// TIA Portal V16 export
// export: Created 2024-05-11T02:56:23.0061867Z, ExportSetting WithDefaults, DisplayName Totally Integrated Automation Portal, DisplayVersion V16, DisplayName TIA Portal Version Control Interface, DisplayVersion V16, DisplayName TIA Portal Openness, DisplayVersion V16, DisplayName STEP 7 Professional, DisplayVersion V16, DisplayName STEP 7 Safety, DisplayVersion V16, DisplayName WinCC Professional, DisplayVersion V16
FUNCTION_BLOCK "F100_Val"   // FB100, LAD
TITLE = 电磁阀控制，
{ S7_Optimized_Access := 'TRUE' }
VERSION : 0.1
// IW_ConMode    00= 双端实际传感器到位，10=出端虚拟到位，11=出双端虚拟到位，01=回端端虚拟到位，
// stored: AutoNumber false, IsIECCheckEnabled false, IsRetainMemResEnabled false, MemoryReserve 100, SetENOAutomatically false, UDAEnableTagReadback false
   VAR_INPUT
      I_AutoAdv : Bool;   // 自动出指令
      I_AutoRet : Bool;   // 自动回指令
      I_ManAdv : Bool;   // 手动出指令
      I_ManRet : Bool;   // 手动回指令
      I_AdvCond : Bool;   // 动作出条件
      I_RetCond : Bool;   // 动作回条件
      I_AdvLS : Bool;   // 伸出到位
      I_RetLS : Bool;   // 返回到位
      IW_AdvTime : Time;   // 出or虚拟延迟
      IW_RetTime : Time;   // 回or虚拟延迟
      IW_AdvTimeOver : Time;   // 伸出超时
      IW_RetTimeOver : Time;   // 返回超时
      I_FoBrRel : Bool;   // 刹车强制解除
      I_Rest : Bool;   // 异常复位
      I_ManMode : Bool;   // 手动模式
      IW_ConMode : UInt;   // 虚拟控制
   END_VAR
   VAR_OUTPUT
      Q_AdvEnd : Bool;   // 伸出到位延迟
      Q_RetEnd : Bool;   // 返回到位延迟
      Q_AdvLS : Bool;   // 伸出到位
      Q_RetLS : Bool;   // 返回到位
      Q_AdvSL : Bool;   // 伸出输出
      Q_RetSL : Bool;   // 返回输出
      Q_FoBraRel : Bool;   // 刹车解除输出
      Q_AdvTiOvErr { ExternalAccessible := 'False'; ExternalVisible := 'False'; ExternalWritable := 'False'} : Bool;   // 出动作超时故障
      Q_RetTiOvErr { ExternalAccessible := 'False'; ExternalVisible := 'False'; ExternalWritable := 'False'} : Bool;   // 回动作超时故障
      Q_SensorsErr : Bool;   // 到位传感器都ON故障
      Q_SenCroErr : Bool;   // 到位传感器交叉ON故障
   END_VAR
   VAR
      MT_AdvChK { ExternalAccessible := 'False'; ExternalVisible := 'False'; ExternalWritable := 'False'} : IEC_TIMER;   // 出端延迟
      MT_RetChK { ExternalAccessible := 'False'; ExternalVisible := 'False'; ExternalWritable := 'False'} : IEC_TIMER;   // 回端延迟
      MT_AdvChKVir { ExternalAccessible := 'False'; ExternalVisible := 'False'; ExternalWritable := 'False'} : IEC_TIMER;   // 出端虚拟延迟
      MT_RetChKVir { ExternalAccessible := 'False'; ExternalVisible := 'False'; ExternalWritable := 'False'} : IEC_TIMER;   // 回端虚拟延迟
      MT_AdvTimeOver { ExternalAccessible := 'False'; ExternalVisible := 'False'; ExternalWritable := 'False'} : IEC_TIMER;   // 出动作延迟
      MT_RetTimeOver { ExternalAccessible := 'False'; ExternalVisible := 'False'; ExternalWritable := 'False'} : IEC_TIMER;   // 回动作延迟
      MT_SenserCrossErro { ExternalAccessible := 'False'; ExternalVisible := 'False'; ExternalWritable := 'False'} : IEC_TIMER;   // 感应器交叉错误判断时间
      M_AdvComm { ExternalAccessible := 'False'; ExternalVisible := 'False'; ExternalWritable := 'False'} : Bool;   // 出动作
      M_RetComm { ExternalAccessible := 'False'; ExternalVisible := 'False'; ExternalWritable := 'False'} : Bool;   // 回动作
   END_VAR
   VAR_TEMP
      M_AdvM : Bool;   // 出指令
      M_RetM : Bool;   // 回指令
      M_SensorsErr : Bool;   // 到位传感器都ON
      M_SenCroErr : Bool;   // 到位传感器交叉ON
   END_VAR
   VAR_TEMP   // added for the SCL form of the ladder/FBD networks
      _w1 : Bool;
   END_VAR
BEGIN

REGION Network 1: 控制指令
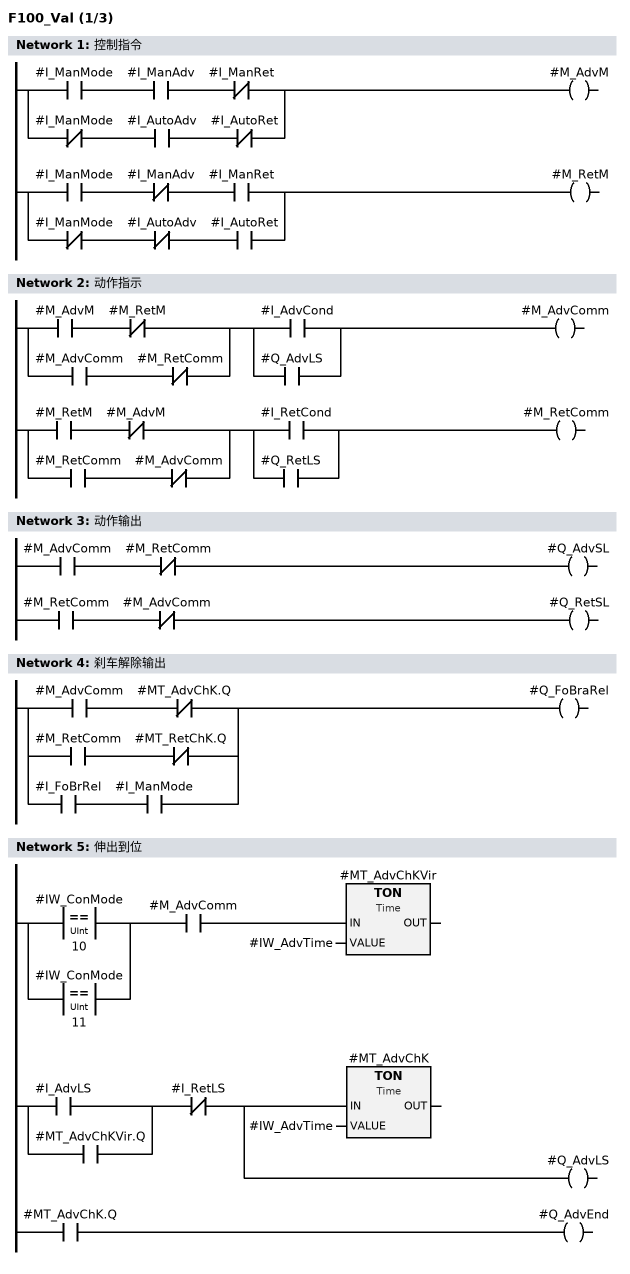
   RUNG wire#powerrail
      Contact( #I_ManMode )
      Contact( #I_ManAdv )
      I_Contact( #I_ManRet )
      wire#w1
      Coil( #M_AdvM )
   END_RUNG
   RUNG wire#powerrail
      I_Contact( #I_ManMode )
      Contact( #I_AutoAdv )
      I_Contact( #I_AutoRet )
   END_RUNG wire#w1
   RUNG wire#powerrail
      Contact( #I_ManMode )
      I_Contact( #I_ManAdv )
      Contact( #I_ManRet )
      wire#w2
      Coil( #M_RetM )
   END_RUNG
   RUNG wire#powerrail
      I_Contact( #I_ManMode )
      I_Contact( #I_AutoAdv )
      Contact( #I_AutoRet )
   END_RUNG wire#w2
   // the same network as SCL:
   #M_AdvM := (#I_ManMode AND #I_ManAdv AND NOT #I_ManRet) OR (NOT #I_ManMode AND #I_AutoAdv AND NOT #I_AutoRet);
   #M_RetM := (#I_ManMode AND NOT #I_ManAdv AND #I_ManRet) OR (NOT #I_ManMode AND NOT #I_AutoAdv AND #I_AutoRet);
END_REGION

REGION Network 2: 动作指示
   RUNG wire#powerrail
      Contact( #M_AdvM )
      I_Contact( #M_RetM )
      wire#w1
      Contact( #I_AdvCond )
      wire#w2
      Coil( #M_AdvComm )
   END_RUNG
   RUNG wire#powerrail
      Contact( #M_AdvComm )
      I_Contact( #M_RetComm )
   END_RUNG wire#w1
   RUNG wire#w1
      Contact( #Q_AdvLS )
   END_RUNG wire#w2
   RUNG wire#powerrail
      Contact( #M_RetM )
      I_Contact( #M_AdvM )
      wire#w3
      Contact( #I_RetCond )
      wire#w4
      Coil( #M_RetComm )
   END_RUNG
   RUNG wire#powerrail
      Contact( #M_RetComm )
      I_Contact( #M_AdvComm )
   END_RUNG wire#w3
   RUNG wire#w3
      Contact( #Q_RetLS )
   END_RUNG wire#w4
   // the same network as SCL:
   #M_AdvComm := ((#M_AdvM AND NOT #M_RetM) OR (#M_AdvComm AND NOT #M_RetComm)) AND (#I_AdvCond OR #Q_AdvLS);
   #M_RetComm := ((#M_RetM AND NOT #M_AdvM) OR (#M_RetComm AND NOT #M_AdvComm)) AND (#I_RetCond OR #Q_RetLS);
END_REGION

REGION Network 3: 动作输出
   RUNG wire#powerrail
      Contact( #M_AdvComm )
      I_Contact( #M_RetComm )
      Coil( #Q_AdvSL )
   END_RUNG
   RUNG wire#powerrail
      Contact( #M_RetComm )
      I_Contact( #M_AdvComm )
      Coil( #Q_RetSL )
   END_RUNG
   // the same network as SCL:
   #Q_AdvSL := #M_AdvComm AND NOT #M_RetComm;
   #Q_RetSL := #M_RetComm AND NOT #M_AdvComm;
END_REGION

REGION Network 4: 刹车解除输出
   RUNG wire#powerrail
      Contact( #M_AdvComm )
      I_Contact( #MT_AdvChK.Q )
      wire#w1
      Coil( #Q_FoBraRel )
   END_RUNG
   RUNG wire#powerrail
      Contact( #M_RetComm )
      I_Contact( #MT_RetChK.Q )
   END_RUNG wire#w1
   RUNG wire#powerrail
      Contact( #I_FoBrRel )
      Contact( #I_ManMode )
   END_RUNG wire#w1
   // the same network as SCL:
   #Q_FoBraRel := (#M_AdvComm AND NOT #MT_AdvChK.Q) OR (#M_RetComm AND NOT #MT_RetChK.Q) OR (#I_FoBrRel AND #I_ManMode);
END_REGION

REGION Network 5: 伸出到位
   #MT_AdvChKVir.TON(IN := ((#IW_ConMode = 10) OR (#IW_ConMode = 11)) AND #M_AdvComm, PT := #IW_AdvTime);   // TON coil
   #_w1 := (#I_AdvLS OR #MT_AdvChKVir.Q) AND NOT #I_RetLS;
   #MT_AdvChK.TON(IN := #_w1, PT := #IW_AdvTime);   // TON coil
   #Q_AdvLS := #_w1;
   #Q_AdvEnd := #MT_AdvChK.Q;
END_REGION

REGION Network 6: 返回到位
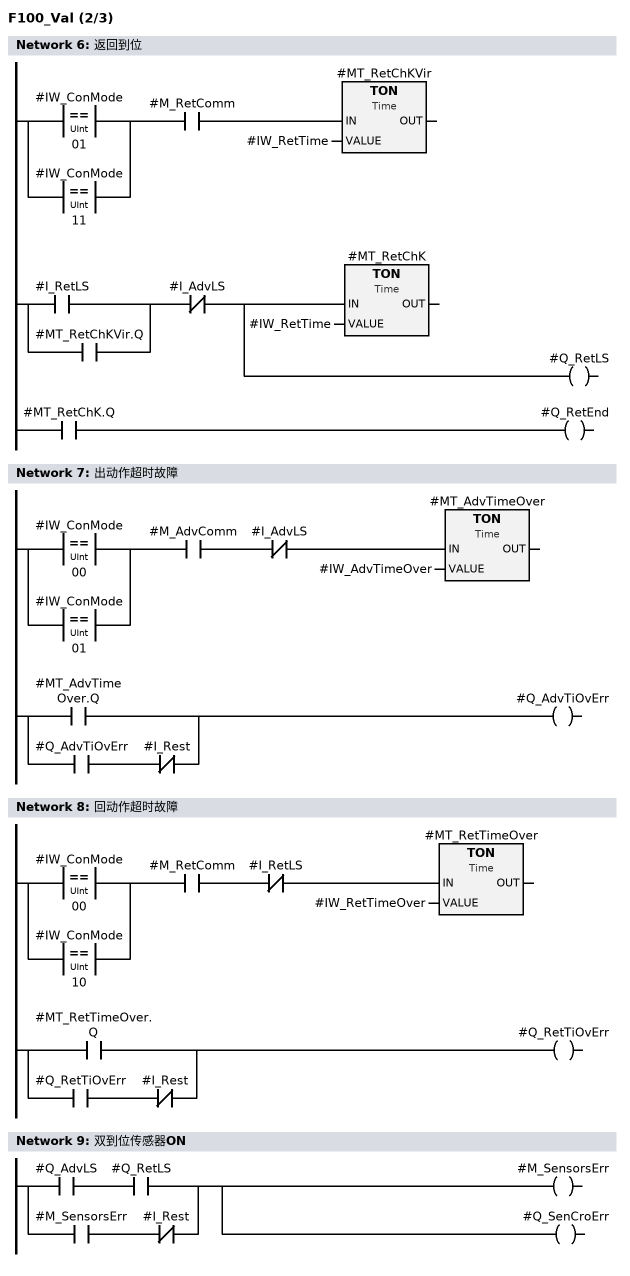
   #MT_RetChKVir.TON(IN := ((#IW_ConMode = 01) OR (#IW_ConMode = 11)) AND #M_RetComm, PT := #IW_RetTime);   // TON coil
   #_w1 := (#I_RetLS OR #MT_RetChKVir.Q) AND NOT #I_AdvLS;
   #MT_RetChK.TON(IN := #_w1, PT := #IW_RetTime);   // TON coil
   #Q_RetLS := #_w1;
   #Q_RetEnd := #MT_RetChK.Q;
END_REGION

REGION Network 7: 出动作超时故障
   #MT_AdvTimeOver.TON(IN := ((#IW_ConMode = 00) OR (#IW_ConMode = 01)) AND #M_AdvComm AND NOT #I_AdvLS, PT := #IW_AdvTimeOver);   // TON coil
   #Q_AdvTiOvErr := #MT_AdvTimeOver.Q OR (#Q_AdvTiOvErr AND NOT #I_Rest);
END_REGION

REGION Network 8: 回动作超时故障
   #MT_RetTimeOver.TON(IN := ((#IW_ConMode = 00) OR (#IW_ConMode = 10)) AND #M_RetComm AND NOT #I_RetLS, PT := #IW_RetTimeOver);   // TON coil
   #Q_RetTiOvErr := #MT_RetTimeOver.Q OR (#Q_RetTiOvErr AND NOT #I_Rest);
END_REGION

REGION Network 9: 双到位传感器ON
   RUNG wire#powerrail
      Contact( #Q_AdvLS )
      Contact( #Q_RetLS )
      wire#w1
      Coil( #M_SensorsErr )
   END_RUNG
   RUNG wire#powerrail
      Contact( #M_SensorsErr )
      I_Contact( #I_Rest )
   END_RUNG wire#w1
   RUNG wire#w1
      Coil( #Q_SenCroErr )
   END_RUNG
   // the same network as SCL:
   #M_SensorsErr := (#Q_AdvLS AND #Q_RetLS) OR (#M_SensorsErr AND NOT #I_Rest);
   #Q_SenCroErr := #M_SensorsErr;
END_REGION

REGION Network 10: 到位传感器交叉ON
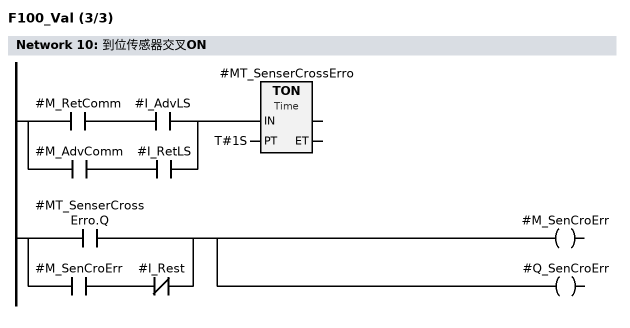
   RUNG wire#powerrail
      Contact( #M_RetComm )
      Contact( #I_AdvLS )
      wire#w1
      { S7_Templates := "time_type := Time" } #MT_SenserCrossErro.TON(pt := T#1S, et =>)
   END_RUNG
   RUNG wire#powerrail
      Contact( #M_AdvComm )
      Contact( #I_RetLS )
   END_RUNG wire#w1
   RUNG wire#powerrail
      Contact( #MT_SenserCrossErro.Q )
      wire#w2
      Coil( #M_SenCroErr )
   END_RUNG
   RUNG wire#powerrail
      Contact( #M_SenCroErr )
      I_Contact( #I_Rest )
   END_RUNG wire#w2
   RUNG wire#w2
      Coil( #Q_SenCroErr )
   END_RUNG
   // the same network as SCL:
   #MT_SenserCrossErro.TON(IN := (#M_RetComm AND #I_AdvLS) OR (#M_AdvComm AND #I_RetLS), PT := T#1S);
   #M_SenCroErr := #MT_SenserCrossErro.Q OR (#M_SenCroErr AND NOT #I_Rest);
   #Q_SenCroErr := #M_SenCroErr;
END_REGION
END_FUNCTION_BLOCK
